// TIA Portal V17 export
// export: Created 2023-10-05T17:26:16.5876413Z, ExportSetting WithDefaults, DisplayName Totally Integrated Automation Portal, DisplayVersion V17, DisplayName TIA Portal Openness, DisplayVersion V17, DisplayName TIA Portal Teamcenter Gateway, DisplayVersion V17, DisplayName TIA Portal Version Control Interface, DisplayVersion V17, DisplayName STEP 7 Professional, DisplayVersion V17, DisplayName STEP 7 Safety, DisplayVersion V17, DisplayName WinCC Advanced / Unified PC, DisplayVersion V17
DATA_BLOCK "Baustein_1_DB"   // DB3
VERSION : 0.1
// stored: AutoNumber true, DBAccessibleFromOPCUA true, InstanceOfName Baustein_1, InstanceOfType FB
"Baustein_1"
   // VAR_OUTPUT
   //    VarB0 : Bool;
   //    VarB1 : Bool;
   //    VarB2 : Bool;
   //    Varb4 : Bool;
   //    VarS1 : Bool;
   // END_VAR
   // VAR_IN_OUT
   //    Test : Bool;
   //    Test2 : Bool;
   // END_VAR
BEGIN
END_DATA_BLOCK
